TYPE ST_System_WT_HWW_Parameter :
STRUCT
	AutoQuittierung			: BOOL ;
END_STRUCT
END_TYPE

(* stored: Version 1.1.0.1, ProductVersion 3.1.4024.9
   DUT ST_System_WT_HWW_Parameter: Id {22783455-1945-40da-91e4-198c50b27db9} *)
